{attribute 'qualified_only'}
VAR_GLOBAL
	// xDI%137.0_A3_2
	MBS_Ref_Taster_DK_Pos_Sauger AT %I*: BOOL;
	// xDI%137.1_A3_2
	MBS_Ref_Taster_DK_Pos_Foerderband AT %I*: BOOL;
	// xDI%137.2_A3_1
	MBS_LS_Ende_Foerderband AT %I*: BOOL;
	// xDI%137.3_A3_2
	MBS_Ref_Taster_DK_Pos_Saege AT %I*: BOOL;
	// xDI%137.4_A3_2
	MBS_Ref_Taster_Sauger_Pos_DK AT %I*: BOOL;
	// xDI%137.5_A3_2
	MBS_Ref_Taster_Ofenschieber_innen AT %I*: BOOL;
	// xDI%137.6_A3_2
	MBS_Ref_Taster_Ofenschieber_aussen AT %I*: BOOL;
	// xDI%137.7_A3_2
	MBS_Ref_Taster_Sauger_Pos_Ofen AT %I*: BOOL;
	// xDI%138.0_A3_1
	MBS_LS_Ofen AT %I*: BOOL;
	// xDO%112.0_A3_4
	MBS_MOT_DK_CW AT %Q*: BOOL;
	// xDO%112.1_A3_4
	MBS_MOT_DK_CCW AT %Q*: BOOL;
	// xDO%112.2_A3_2
	MBS_MOT_Foerderband_vorwaerts AT %Q*: BOOL;
	// xDO%112.3_A3_6
	MBS_MOT_Saege AT %Q*: BOOL;
	// xDO%112.4_A3_3
	MBS_MOT_Ofenschieber_einfahren AT %Q*: BOOL;
	// xDO%112.5_A3_3
	MBS_MOT_Ofenschieber_ausfahren AT %Q*: BOOL;
	// xDO%112.6_A3_5
	MBS_MOT_Sauger_zum_Ofen AT %Q*: BOOL;
	// xDO%112.7_A3_5
	MBS_MOT_Sauger_zum_DK AT %Q*: BOOL;
	// xDO%113.0_A3_7
	MBS_Leuchte_Ofen AT %Q*: BOOL;
	// xDO%113.1_A3_8
	MBS_Kompressor AT %Q*: BOOL;
	// xDO%113.2_A3_5
	MBS_MV_Vakuum AT %Q*: BOOL;
	// xDO%113.3_A3_5
	MBS_MV_senken AT %Q*: BOOL;
	// xDO%113.4_A3_5
	MBS_MV_Ofentuer AT %Q*: BOOL;
	// xDO%113.5_A3_5
	MBS_MV_Schieber AT %Q*: BOOL;
END_VAR

(* stored: Version 1.1.0.1, ProductVersion 3.1.4024.15
   GVL GVL_MBS: Id {2884d7c7-6a6f-4ec2-a6e8-4dfa5604880f} *)
